FUNCTION_BLOCK ProfiNetMaster
VAR_INPUT
END_VAR
VAR_OUTPUT
END_VAR
VAR
	DevState AT%I* : UINT;
	PnIoError AT%I* : UINT;
	PnIoDiag AT%i* : UINT;
END_VAR

END_FUNCTION_BLOCK

(* stored: Version 1.1.0.1, ProductVersion 3.1.4024.11
   POU ProfiNetMaster: Id {1b53501a-4658-47c6-ac20-372be2f8e652}, SpecialFunc None *)
